// TIA Portal V16 export
// export: Created 2024-05-10T06:46:43.9188795Z, ExportSetting WithDefaults, DisplayName Totally Integrated Automation Portal, DisplayVersion V16, DisplayName TIA Portal Version Control Interface, DisplayVersion V16, DisplayName TIA Portal Openness, DisplayVersion V16, DisplayName STEP 7 Professional, DisplayVersion V16, DisplayName STEP 7 Safety, DisplayVersion V16, DisplayName WinCC Professional, DisplayVersion V16
DATA_BLOCK "K19_ST07上自动_DB"   // DB19
VERSION : 0.1
// stored: AutoNumber false, DBAccessibleFromOPCUA true, InstanceOfName K19_ST07上自动, InstanceOfType FB
"K19_ST07上自动"
BEGIN
END_DATA_BLOCK
